{attribute 'GeneratedUsingTerminal: EL3483-0000-0016'}
{attribute addProperty BoxType "EL3483-0000-0016"}
{attribute addProperty Id "L1_StatusAT %I*L1_Status_12B1E6BB5L2_StatusAT %I*L2_Status_12B1E6BB5L3_StatusAT %I*L3_Status_12B1E6BB5Total_StatusAT %I*Total_Status_AD43C3B912Total_AdvancedAT %I*Total_Advanced_3B87F4672WcStateAT %I*WcState_9091E0EB2InfoDataAT %I*InfoData_94A18F5E2"}
{attribute addProperty CRC "37282642"}
{attribute addProperty Size "33"}
TYPE EL3483_0238E352 EXTENDS EtcSlaveTerminalBase_947E5A46 :
STRUCT
	{attribute addProperty Name "L1_Status"}
	L1_Status : L1_Status_12B1E6BB;
	{attribute addProperty Name "L2_Status"}
	L2_Status : L2_Status_12B1E6BB;
	{attribute addProperty Name "L3_Status"}
	L3_Status : L3_Status_12B1E6BB;
	{attribute addProperty Name "Total_Status"}
	Total_Status : Total_Status_AD43C3B9;
	{attribute addProperty Name "Total_Advanced"}
	Total_Advanced : Total_Advanced_3B87F467;
	{attribute addProperty Name "WcState"}
	WcState : WcState_9091E0EB;
	{attribute addProperty Name "InfoData"}
	InfoData : InfoData_94A18F5E;
END_STRUCT
END_TYPE

(* stored: Version 1.2.0.0, ProductVersion 3.1.4024.9
   DUT EL3483_0238E352: Id {821df97b-014c-43f8-9771-9175334cf171} *)
